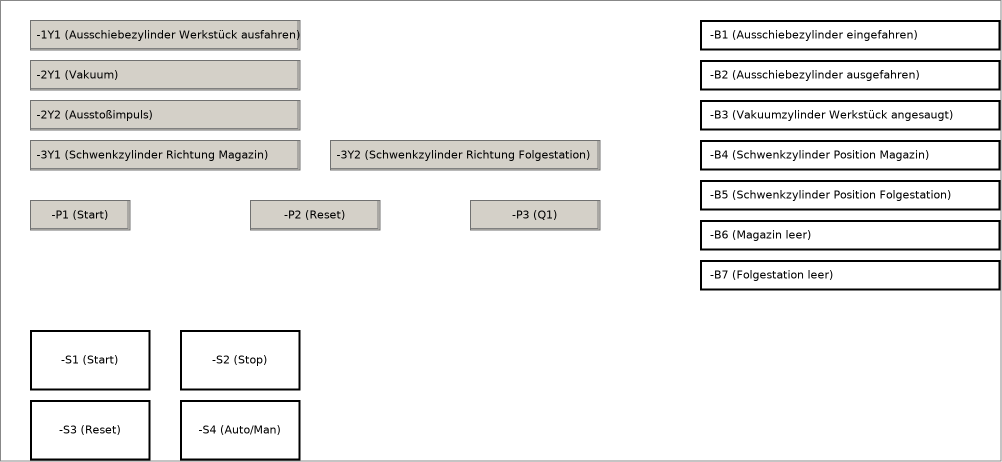
VISUALIZATION MPS_Station_Verteilen  // 1002x462
    Button (30,200 100x30), "-P1 (Start)"
        tap dSub.P1
    Button (250,200 130x30), "-P2 (Reset)"
        tap dSub.P2
    Button (470,200 130x30), "-P3 (Q1)"
        tap dSub.P3
    Button (30,20 270x30), "-1Y1 (Ausschiebezylinder Werkstück ausfahren)"
        tap dSub.Y1_1
    Rectangle (30,330 120x60), "-S1 (Start)", colour toggle: dSub.S1
    Rectangle (180,330 120x60), "-S2 (Stop)", colour toggle: dSub.S2
    Rectangle (30,400 120x60), "-S3 (Reset)", colour toggle: dSub.S4
    Rectangle (180,400 120x60), "-S4 (Auto/Man)", colour toggle: dSub.S3
    Rectangle (700,20 300x30), "-B1 (Ausschiebezylinder eingefahren)", colour toggle: dSub.B1
    Rectangle (700,60 300x30), "-B2 (Ausschiebezylinder ausgefahren)", colour toggle: dSub.B2
    Rectangle (700,100 300x30), "-B3 (Vakuumzylinder Werkstück angesaugt)", colour toggle: dSub.B3
    Rectangle (700,140 300x30), "-B4 (Schwenkzylinder Position Magazin)", colour toggle: dSub.B4
    Rectangle (700,180 300x30), "-B5 (Schwenkzylinder Position Folgestation)", colour toggle: dSub.B5
    Rectangle (700,220 300x30), "-B6 (Magazin leer)", colour toggle: dSub.B6
    Rectangle (700,260 300x30), "-B7 (Folgestation leer)", colour toggle: dSub.B7
    Button (30,60 270x30), "-2Y1 (Vakuum)"
        tap dSub.Y2_1
    Button (30,100 270x30), "-2Y2 (Ausstoßimpuls)"
        tap dSub.Y2_2
    Button (30,140 270x30), "-3Y1 (Schwenkzylinder Richtung Magazin)"
        tap dSub.Y3_1
    Button (330,140 270x30), "-3Y2 (Schwenkzylinder Richtung Folgestation)"
        tap dSub.Y3_2
END_VISUALIZATION

(* stored: Version 1.1.0.1, ProductVersion 3.1.4022.6
   Visu MPS_Station_Verteilen: Id {529ab607-a3a7-4016-be48-cafee3caa910} *)
